FUNCTION_BLOCK BFB_GPIO
  (* Standard: 61499-2 *)
  (* Version 0.1, 2016-00-31, hpea485, UOA *)
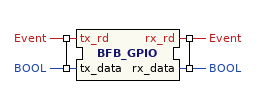
  EVENT_INPUT
    tx_rd WITH tx_data;
  END_EVENT
  EVENT_OUTPUT
    rx_rd WITH rx_data;
  END_EVENT
  VAR_INPUT
    tx_data : BOOL;
  END_VAR
  VAR_OUTPUT
    rx_data : BOOL;
  END_VAR
  VAR
    tx_gpio : BOOL; (* TOPIO_OUT *)
    rx_gpio : BOOL; (* TOPIO_IN *)
  END_VAR
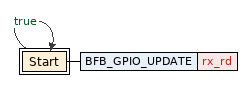
  EC_STATES
    Start : BFB_GPIO_UPDATE -> rx_rd;
  END_STATES
  EC_TRANSITIONS
    Start TO Start := true;
  END_TRANSITIONS
  ALGORITHM BFB_GPIO_UPDATE IN VHDL:
rx_data <= rx_gpio;
tx_gpio <= tx_data;
DONE <= '1';
  END_ALGORITHM
END_FUNCTION_BLOCK
